PROGRAM MAIN
VAR
END_VAR

ACTION StartStopMotor:
// NETWORK 1
END_ACTION

END_PROGRAM

(* stored: Version 1.1.0.1, ProductVersion 3.1.4024.12
   POU MAIN: Id {6ef22546-1438-4d6e-9651-886b4f55e901}, SpecialFunc None
   Action StartStopMotor: Id {62300328-5c8e-4ad3-9294-7de29600394f} *)
